FUNCTION F_InitializeAllElements :BOOL
(**************************************************************************************
 * 	Application		:	BoxControl Framework
 *	Revision		:	$Revision: 404529 $
 *	Revision date	:	$Date: 2018-04-23 08:21:38 +0200 (Mo., 23 Apr 2018) $
 *	Last changed by	:	$Author: b7bolm $
 *	URL				:	$URL: http://almscdc.swisslog.com/repo/SWPD/Development/BoxControlFramework/20_Release/trunk/01_Software/BCF/BCF/JumpStart/20_Product/10_App/13_Elements/10_Lib/10_Conv/10_Functions/F_InitializeAllElements.TcPOU $
 *
 *	Purpose			:	Initialize all elements
 *
 * ------------------------------------------------------------------------------------
 *	Copyright Swisslog [IP AG], Switzerland. All rights reserved.
 * 
 * ------------------------------------------------------------------------------------
 *	
 * 	Revision History: 
 *
 * 	VERSION			DATE			INITIALS			DESCRIPTION
 *	0.1				01.01.2001		swl					Example
 *
 **************************************************************************************)
VAR
	eElementNumber		: E_ElementNumber; // Element number
END_VAR


// Loop over all elements and initialize each element 
FOR eElementNumber := E_ElementNumber.E_BEGIN_ELEMENT+ 1 TO E_ElementNumber.E_END_ELEMENT- 1 DO
	// If reference is valid
	IF __ISVALIDREF(ElementRegistry[eElementNumber].rElement) THEN
		// Initialize element
		ElementRegistry[eElementNumber].rElement.M_InitElement(TRUE);
	END_IF
END_FOR

END_FUNCTION

(* stored: Version 1.1.0.1, ProductVersion 3.1.4022.12
   POU F_InitializeAllElements: Id {ae6f90de-e2ef-47ee-84aa-82a63935aa22}, SpecialFunc None *)
